	(* Internal method *)
	{attribute 'hide'}
	METHOD FB_init : BOOL
	VAR_INPUT
		(*  if TRUE, the retain variables are initialized (warm start / cold start) *)
		bInitRetains : BOOL;
		(*  if TRUE, the instance afterwards gets moved into the copy code (online change) *)
		bInCopyCode : BOOL;
	END_VAR
END_METHOD


	(* Internal method *)
	{attribute 'hide'}
	METHOD FB_exit : BOOL
	VAR_INPUT
		(*  if TRUE, the exit method is called for exiting an instance that is copied afterwards (online change). *)
		bInCopyCode : BOOL;
	END_VAR
END_METHOD


	(* Set the rotation angle in degrees [Â°]. *)
	METHOD SetAngle
	VAR_INPUT
		(* Rotation angle to set in degrees [Â°]. *)
		angle : LREAL;
	END_VAR
END_METHOD


	(* Set the components of this vector to '0.0'. *)
	METHOD SetZero
END_METHOD


	(* Set the components of this orientation. *)
	METHOD SetValues
	VAR_IN_OUT
		(* The position values to set. *)
 {attribute 'GUID' := '9769C204-E8C9-2F95-61E1-FD1671A2860B'}
				orientation2D : Orientation2D;
	END_VAR
END_METHOD


	(* Get the direction of the local x-axis. *)
	METHOD GetDirectionX
	VAR_IN_OUT
		(* The local x-direction of this orientation. *)
 {attribute 'GUID' := '5D3BC02D-EA16-22EA-7ADA-76A9B505DC98'}
				localX : TangentXY;
	END_VAR
END_METHOD


	(* Get the direction of the local y-axis. *)
	METHOD GetDirectionY
	VAR_IN_OUT
		(* The local y-direction of this orientation. *)
 {attribute 'GUID' := '5D3BC02D-EA16-22EA-7ADA-76A9B505DC98'}
				localY : TangentXY;
	END_VAR
END_METHOD


	(* Invert this position. *)
	METHOD Invert
END_METHOD


	(* Multiply an orientation to this orientation. *)
	METHOD ConcatenateWith
	VAR_IN_OUT
		(* Orientation to concatenate with. *)
 {attribute 'GUID' := '9769C204-E8C9-2F95-61E1-FD1671A2860B'}
				orientation2D : Orientation2D;
	END_VAR
END_METHOD


	(* Turn the orientation. *)
	METHOD TurnByC
	VAR_INPUT
		(* Rotation angle to turn by in degrees [Â°]. *)
		angle : LREAL;
	END_VAR
END_METHOD


	(* Rotate a PositionXY according to this orientation. *)
	METHOD Transform
	VAR_IN_OUT
		(* The orientation to multipy by. *)
 {attribute 'GUID' := 'ED71C9D8-8E4B-28CC-7DA0-249C4B114DE7'}
				positionXY : PositionXY;
	END_VAR
END_METHOD


	PROPERTY angle : LREAL
GET
END_GET
SET
END_SET
END_PROPERTY

END_FUNCTION_BLOCK

// POUs/Spatial/Functions/ConcatenateABC

	{attribute 'TcIecLibraryType'}
	{attribute 'external_name' := 'ConcatenateABC_GUID_63EF3EFF_CE46_22F7_7592_D84453B7BE61'}
	(* Concatenate two instances of Orientation3D. *)
	FUNCTION ConcatenateABC : BOOL
	VAR_IN_OUT
		rotation0	:	Orientation3D;	(* 1st input orientation of the concatenation. *)
		rotation1	:	Orientation3D;	(* 2nd input orientation of the concatenation. *)
		concatenation	:	Orientation3D;	(* The concatenation of the two input instances. *)
	END_VAR

END_FUNCTION

// POUs/Spatial/Positions/Orientation3D

	{attribute 'c++_compatible'}
	{attribute 'external_name' := 'Orientation3D_GUID_F3A50331_CB69_26F7_728F_6AA10FEBE6C7'}
	{attribute 'TcIecLibraryType'}
	{attribute 'no_explicit_call' :='do not call this POU directly'}
	{attribute 'no_assign'}
	(* 3D orientation. All angles in degrees [Â°]. *)
	FUNCTION_BLOCK Orientation3D
	VAR
		(* Rotation around the 1st local axis in degrees [Â°]. *)
		p0 : LREAL;
		(* Rotation around 2nd local axis in degrees [Â°]. *)
		p1 : LREAL;
		(* Rotation around 3rd local axis in degrees [Â°]. *)
		p2 : LREAL;
		(* Defines the rotation order (rotate around local axes from left to right) *)
		 {attribute 'GUID' := 'BF8BCC1E-925E-4A57-801C-CC42AFDDA86D'}
		coordinates : E_RotationCoordinates := E_RotationCoordinates.CBA;
		 {attribute 'hide'}
		_reserved1 : ARRAY [1..84] OF USINT;
	END_VAR


	(* Internal method *)
	{attribute 'hide'}
	METHOD FB_init : BOOL
	VAR_INPUT
		(*  if TRUE, the retain variables are initialized (warm start / cold start) *)
		bInitRetains : BOOL;
		(*  if TRUE, the instance afterwards gets moved into the copy code (online change) *)
		bInCopyCode : BOOL;
	END_VAR
END_METHOD


	(* Internal method *)
	{attribute 'hide'}
	METHOD FB_exit : BOOL
	VAR_INPUT
		(*  if TRUE, the exit method is called for exiting an instance that is copied afterwards (online change). *)
		bInCopyCode : BOOL;
	END_VAR
END_METHOD


	(* Set the components of this vector to '0.0'. *)
	METHOD SetZero
END_METHOD


	(* Set the components of this position. *)
	METHOD SetValues
	VAR_IN_OUT
		(* The position values to set. *)
 {attribute 'GUID' := 'F3A50331-CB69-26F7-728F-6AA10FEBE6C7'}
				orientation3D : Orientation3D;
	END_VAR
END_METHOD


	(* Set the coordinates of the orientation. *)
	METHOD SetValuesABC
	VAR_INPUT
		(* 1st rotation angle in degrees [Â°]. *)
		phi0 : LREAL;
		(* 2nd rotation angle in degrees [Â°]. *)
		phi1 : LREAL;
		(* 3rd rotation angle in degrees [Â°]. *)
		phi2 : LREAL;
	END_VAR
END_METHOD


	(* Set the coordinates of the orientation. *)
	METHOD SetValuesACB
	VAR_INPUT
		(* 1st rotation angle in degrees [Â°]. *)
		phi0 : LREAL;
		(* 2nd rotation angle in degrees [Â°]. *)
		phi1 : LREAL;
		(* 3rd rotation angle in degrees [Â°]. *)
		phi2 : LREAL;
	END_VAR
END_METHOD


	(* Set the coordinates of the orientation. *)
	METHOD SetValuesBCA
	VAR_INPUT
		(* 1st rotation angle in degrees [Â°]. *)
		phi0 : LREAL;
		(* 2nd rotation angle in degrees [Â°]. *)
		phi1 : LREAL;
		(* 3rd rotation angle in degrees [Â°]. *)
		phi2 : LREAL;
	END_VAR
END_METHOD


	(* Set the coordinates of the orientation. *)
	METHOD SetValuesBAC
	VAR_INPUT
		(* 1st rotation angle in degrees [Â°]. *)
		phi0 : LREAL;
		(* 2nd rotation angle in degrees [Â°]. *)
		phi1 : LREAL;
		(* 3rd rotation angle in degrees [Â°]. *)
		phi2 : LREAL;
	END_VAR
END_METHOD


	(* Set the coordinates of the orientation. *)
	METHOD SetValuesCAB
	VAR_INPUT
		(* 1st rotation angle in degrees [Â°]. *)
		phi0 : LREAL;
		(* 2nd rotation angle in degrees [Â°]. *)
		phi1 : LREAL;
		(* 3rd rotation angle in degrees [Â°]. *)
		phi2 : LREAL;
	END_VAR
END_METHOD


	(* Set the coordinates of the orientation. *)
	METHOD SetValuesCBA
	VAR_INPUT
		(* 1st rotation angle in degrees [Â°]. *)
		phi0 : LREAL;
		(* 2nd rotation angle in degrees [Â°]. *)
		phi1 : LREAL;
		(* 3rd rotation angle in degrees [Â°]. *)
		phi2 : LREAL;
	END_VAR
END_METHOD


	(* Set the coordinates of the orientation. *)
	METHOD SetValuesABA
	VAR_INPUT
		(* 1st rotation angle in degrees [Â°]. *)
		phi0 : LREAL;
		(* 2nd rotation angle in degrees [Â°]. *)
		phi1 : LREAL;
		(* 3rd rotation angle in degrees [Â°]. *)
		phi2 : LREAL;
	END_VAR
END_METHOD


	(* Set the coordinates of the orientation. *)
	METHOD SetValuesACA
	VAR_INPUT
		(* 1st rotation angle in degrees [Â°]. *)
		phi0 : LREAL;
		(* 2nd rotation angle in degrees [Â°]. *)
		phi1 : LREAL;
		(* 3rd rotation angle in degrees [Â°]. *)
		phi2 : LREAL;
	END_VAR
END_METHOD


	(* Set the coordinates of the orientation. *)
	METHOD SetValuesBCB
	VAR_INPUT
		(* 1st rotation angle in degrees [Â°]. *)
		phi0 : LREAL;
		(* 2nd rotation angle in degrees [Â°]. *)
		phi1 : LREAL;
		(* 3rd rotation angle in degrees [Â°]. *)
		phi2 : LREAL;
	END_VAR
END_METHOD


	(* Set the coordinates of the orientation. *)
	METHOD SetValuesBAB
	VAR_INPUT
		(* 1st rotation angle in degrees [Â°]. *)
		phi0 : LREAL;
		(* 2nd rotation angle in degrees [Â°]. *)
		phi1 : LREAL;
		(* 3rd rotation angle in degrees [Â°]. *)
		phi2 : LREAL;
	END_VAR
END_METHOD


	(* Set the coordinates of the orientation. *)
	METHOD SetValuesCAC
	VAR_INPUT
		(* 1st rotation angle in degrees [Â°]. *)
		phi0 : LREAL;
		(* 2nd rotation angle in degrees [Â°]. *)
		phi1 : LREAL;
		(* 3rd rotation angle in degrees [Â°]. *)
		phi2 : LREAL;
	END_VAR
END_METHOD


	(* Set the coordinates of the orientation. *)
	METHOD SetValuesCBC
	VAR_INPUT
		(* 1st rotation angle in degrees [Â°]. *)
		phi0 : LREAL;
		(* 2nd rotation angle in degrees [Â°]. *)
		phi1 : LREAL;
		(* 3rd rotation angle in degrees [Â°]. *)
		phi2 : LREAL;
	END_VAR
END_METHOD


	(* Get the direction of the local x-axis. *)
	METHOD GetDirectionX
	VAR_IN_OUT
		(* The local x-direction of this orientation. *)
 {attribute 'GUID' := '8E451EF0-1EF7-2C22-40FE-C3C408FD9C3F'}
				localX : Tangent3D;
	END_VAR
END_METHOD


	(* Get the direction of the local y-axis. *)
	METHOD GetDirectionY
	VAR_IN_OUT
		(* The local y-direction of this orientation. *)
 {attribute 'GUID' := '8E451EF0-1EF7-2C22-40FE-C3C408FD9C3F'}
				localY : Tangent3D;
	END_VAR
END_METHOD


	(* Get the direction of the local z-axis. *)
	METHOD GetDirectionZ
	VAR_IN_OUT
		(* The local z-direction of this orientation. *)
 {attribute 'GUID' := '8E451EF0-1EF7-2C22-40FE-C3C408FD9C3F'}
				localZ : Tangent3D;
	END_VAR
END_METHOD


	(* Invert this position. *)
	METHOD Invert
END_METHOD


	(* Multiply an orientation to this orientation. *)
	METHOD ConcatenateWith
	VAR_IN_OUT
		(* Orientation to concatenate with. *)
 {attribute 'GUID' := 'F3A50331-CB69-26F7-728F-6AA10FEBE6C7'}
				orientation : Orientation3D;
	END_VAR
END_METHOD


	(* Rotate around an arbitrary local axis. The turn angle is given by the length of the axis. *)
	METHOD TurnBy
	VAR_IN_OUT
		(* The axis of rotation. Its length represents the angle of rotation in degrees [Â°]. *)
 {attribute 'GUID' := '7C1DEECE-32AB-2E94-7A82-2C8AD444717E'}
				axis : TangentABC;
	END_VAR
END_METHOD


	(* Rotation around the local x-axis. *)
	METHOD TurnByA
	VAR_INPUT
		(* The angle to rotate by in degrees [Â°]. *)
		da : LREAL;
	END_VAR
END_METHOD


	(* Rotation around the local y-axis. *)
	METHOD TurnByB
	VAR_INPUT
		(* The angle to rotate by in degrees [Â°]. *)
		db : LREAL;
	END_VAR
END_METHOD


	(* Rotation around the local z-axis. *)
	METHOD TurnByC
	VAR_INPUT
		(* The angle to rotate by in degrees [Â°]. *)
		dc : LREAL;
	END_VAR
END_METHOD


	(* Rotate a Position3D according to this orientation. *)
	METHOD Transform
	VAR_IN_OUT
		(* Position to transform. *)
 {attribute 'GUID' := '513B7ECA-E1D5-262C-5763-788E1FD4F5AD'}
				position3D : Position3D;
	END_VAR
END_METHOD


	PROPERTY phi0 : LREAL
GET
END_GET
SET
END_SET
END_PROPERTY


	PROPERTY phi1 : LREAL
GET
END_GET
SET
END_SET
END_PROPERTY


	PROPERTY phi2 : LREAL
GET
END_GET
SET
END_SET
END_PROPERTY


	PROPERTY convention : E_RotationCoordinates
GET
END_GET
SET
END_SET
END_PROPERTY

END_FUNCTION_BLOCK

// POUs/Spatial/Functions/ConcatenateXYC

	{attribute 'TcIecLibraryType'}
	{attribute 'external_name' := 'ConcatenateXYC_GUID_447068A6_9467_2251_75A9_C1FF62E2E084'}
	(* Concatenate two instances of PositionXYC. *)
	FUNCTION ConcatenateXYC : BOOL
	VAR_IN_OUT
		position0	:	PositionXYC;	(* 1st input position of the concatenation. *)
		position1	:	PositionXYC;	(* 2nd input position of the concatenation. *)
		concatenation	:	PositionXYC;	(* The concatenation of the two input instances. *)
	END_VAR

END_FUNCTION

// POUs/Spatial/Functions/Concatenate6D

	{attribute 'TcIecLibraryType'}
	{attribute 'external_name' := 'Concatenate6D_GUID_B218722C_9A1D_2627_473C_2033807B3EB5'}
	(* Concatenate two instances of PositionSE3. *)
	FUNCTION Concatenate6D : BOOL
	VAR_IN_OUT
		position0	:	PositionSE3;	(* 1st input position of the concatenation. *)
		position1	:	PositionSE3;	(* 2nd input position of the concatenation. *)
		concatenation	:	PositionXYC;	(* The concatenation of the two input instances. *)
	END_VAR

END_FUNCTION

// POUs/Spatial/Functions/AddXY

	{attribute 'TcIecLibraryType'}
	{attribute 'external_name' := 'AddXY_GUID_E175C5D9_61B7_2C72_416A_96A339F4B43B'}
	(* Add two instances of TangentXY. *)
	FUNCTION AddXY : BOOL
	VAR_IN_OUT
		tangent0	:	TangentXY;	(* 1st input tangent vector. *)
		tangent1	:	TangentXY;	(* 2nd input tangent vector. *)
		sumTangent	:	TangentXY;	(* Sum of the two tangent vectors. *)
	END_VAR

END_FUNCTION

// POUs/Spatial/Functions/SubtractXY

	{attribute 'TcIecLibraryType'}
	{attribute 'external_name' := 'SubtractXY_GUID_30C9C628_6AA3_2EA8_7056_6D631FEDD6CC'}
	(* Subtract two instances of TangentXY. *)
	FUNCTION SubtractXY : BOOL
	VAR_IN_OUT
		tangent0	:	TangentXY;	(* 1st input tangent vector. *)
		tangent1	:	TangentXY;	(* 2nd input tangent vector. *)
		difference	:	TangentXY;	(* Difference of the two tangent vectors. *)
	END_VAR

END_FUNCTION

// POUs/Spatial/Functions/MultiplyXY

	{attribute 'TcIecLibraryType'}
	{attribute 'external_name' := 'MultiplyXY_GUID_FE62303C_7D56_2E0D_77DF_EC3A00A94E9C'}
	(* Multiply a TangentXY by a scalar and return the result. *)
	FUNCTION MultiplyXY : BOOL
	VAR_IN_OUT
		tangent	:	TangentXY;	(* Tangent vector to multiply. *)
	END_VAR
	VAR_INPUT
		scalar	:	LREAL;	(* Scalar value to multiply with. *)
	END_VAR
	VAR_IN_OUT
		scaled	:	TangentXY;	(* Scaled input tangent vector. *)
	END_VAR

END_FUNCTION

// POUs/Spatial/Functions/ScalarXY

	{attribute 'TcIecLibraryType'}
	{attribute 'external_name' := 'ScalarXY_GUID_E87FF040_9366_28D4_7F75_DB012A742D5B'}
	(* Compute the scalar product of two instance of TangentXY. *)
	FUNCTION ScalarXY : LREAL
	VAR_IN_OUT
		tangent0	:	TangentXY;	(* 1st input tangent vector. *)
		tangent1	:	TangentXY;	(* 2nd input tangent vector. *)
	END_VAR

END_FUNCTION

// POUs/Spatial/Functions/Add3D

	{attribute 'TcIecLibraryType'}
	{attribute 'external_name' := 'Add3D_GUID_22B5713A_DAAE_208F_5845_FFB0DA8961E0'}
	(* Add two instances of Tangent3D. *)
	FUNCTION Add3D : BOOL
	VAR_IN_OUT
		tangent0	:	Tangent3D;	(* 1st input tangent vector. *)
		tangent1	:	Tangent3D;	(* 2nd input tangent vector. *)
		sumTangent	:	Tangent3D;	(* Sum of the two tangent vectors. *)
	END_VAR

END_FUNCTION

// POUs/Spatial/Functions/Subtract3D

	{attribute 'TcIecLibraryType'}
	{attribute 'external_name' := 'Subtract3D_GUID_3F13D96E_61B4_2521_768F_ABB3A2BB8B32'}
	(* Subtract two instances of Tangent3D. *)
	FUNCTION Subtract3D : BOOL
	VAR_IN_OUT
		tangent0	:	Tangent3D;	(* 1st input tangent vector. *)
		tangent1	:	Tangent3D;	(* 2nd input tangent vector. *)
		difference	:	Tangent3D;	(* Difference of the two tangent vectors. *)
	END_VAR

END_FUNCTION

// POUs/Spatial/Functions/Multiply3D

	{attribute 'TcIecLibraryType'}
	{attribute 'external_name' := 'Multiply3D_GUID_43B67DFD_6BDE_217D_78F1_09963C777F30'}
	(* Multiply a Tangent3D by a scalar. *)
	FUNCTION Multiply3D : BOOL
	VAR_IN_OUT
		tangent	:	Tangent3D;	(* Tangent vector to multiply. *)
	END_VAR
	VAR_INPUT
		scalar	:	LREAL;	(* Scalar value to multiply with. *)
	END_VAR
	VAR_IN_OUT
		scaled	:	Tangent3D;	(* Scaled input tangent vector. *)
	END_VAR

END_FUNCTION

// POUs/Spatial/Functions/Scalar3D

	{attribute 'TcIecLibraryType'}
	{attribute 'external_name' := 'Scalar3D_GUID_B656DD08_36BC_2264_65B8_8E86D53E44D8'}
	(* Compute the scalar product of two instances of Tangent3D. *)
	FUNCTION Scalar3D : LREAL
	VAR_IN_OUT
		tangent0	:	Tangent3D;	(* 1st input tangent vector. *)
		tangent1	:	Tangent3D;	(* 2nd input tangent vector. *)
	END_VAR

END_FUNCTION

// POUs/Spatial/Functions/Cross3D

	{attribute 'TcIecLibraryType'}
	{attribute 'external_name' := 'Cross3D_GUID_637E2F8F_7C67_21A9_5D9B_C69EDB5530E5'}
	(* Compute the cross product of two instances of Tangent3D. *)
	FUNCTION Cross3D : BOOL
	VAR_IN_OUT
		tangent0	:	Tangent3D;	(* 1st input tangent vector. *)
		tangent1	:	Tangent3D;	(* 2nd input tangent vector. *)
		crossProduct	:	Tangent3D;	(* The resulting cross product. *)
	END_VAR

END_FUNCTION

// POUs/Spatial/Functions/AddABC

	{attribute 'TcIecLibraryType'}
	{attribute 'external_name' := 'AddABC_GUID_B378EB54_DC30_2FB7_4703_748A68BC554E'}
	(* Add two instances of TangentABC. *)
	FUNCTION AddABC : BOOL
	VAR_IN_OUT
		tangent0	:	TangentABC;	(* 1st input tangent vector. *)
		tangent1	:	TangentABC;	(* 2nd input tangent vector. *)
		sumTangent	:	TangentABC;	(* Sum of the two tangent vectors. *)
	END_VAR

END_FUNCTION

// POUs/Spatial/Functions/SubtractABC

	{attribute 'TcIecLibraryType'}
	{attribute 'external_name' := 'SubtractABC_GUID_0EC77355_F7D6_2D64_72F6_4550677466CB'}
	(* Subtract two instances of TangentABC. *)
	FUNCTION SubtractABC : BOOL
	VAR_IN_OUT
		tangent0	:	TangentABC;	(* 1st input tangent vector. *)
		tangent1	:	TangentABC;	(* 2nd input tangent vector. *)
		difference	:	TangentABC;	(* Difference of the two tangent vectors. *)
	END_VAR

END_FUNCTION

// POUs/Spatial/Functions/MultiplyABC

	{attribute 'TcIecLibraryType'}
	{attribute 'external_name' := 'MultiplyABC_GUID_CED5725A_0908_2221_656C_470734809FE5'}
	(* Multiply a TangentABC by a scalar. *)
	FUNCTION MultiplyABC : BOOL
	VAR_IN_OUT
		tangent	:	TangentABC;	(* Tangent vector to multiply. *)
	END_VAR
	VAR_INPUT
		scalar	:	LREAL;	(* Scalar value to multiply with. *)
	END_VAR
	VAR_IN_OUT
		scaled	:	TangentABC;	(* Scaled input tangent vector. *)
	END_VAR

END_FUNCTION

// POUs/Spatial/Functions/AddXYC

	{attribute 'TcIecLibraryType'}
	{attribute 'external_name' := 'AddXYC_GUID_1E14462F_988B_29BB_78EF_085C7340C86C'}
	(* Add two instances of TangentXYC. *)
	FUNCTION AddXYC : BOOL
	VAR_IN_OUT
		tangent0	:	TangentXYC;	(* 1st input tangent vector. *)
		tangent1	:	TangentXYC;	(* 2nd input tangent vector. *)
		sumTangent	:	TangentXYC;	(* Sum of the two tangent vectors. *)
	END_VAR

END_FUNCTION

// POUs/Spatial/Functions/SubtractXYC

	{attribute 'TcIecLibraryType'}
	{attribute 'external_name' := 'SubtractXYC_GUID_DDE910B0_CB45_27E1_47FA_8B6FC171A22B'}
	(* Subtract two instances of TangentXYC. *)
	FUNCTION SubtractXYC : BOOL
	VAR_IN_OUT
		tangent0	:	TangentXYC;	(* 1st input tangent vector. *)
		tangent1	:	TangentXYC;	(* 2nd input tangent vector. *)
		difference	:	TangentXYC;	(* Difference of the two tangent vectors. *)
	END_VAR

END_FUNCTION

// POUs/Spatial/Functions/MultiplyXYC

	{attribute 'TcIecLibraryType'}
	{attribute 'external_name' := 'MultiplyXYC_GUID_6B3384A2_CB86_2C92_42CE_70FAA85DA471'}
	(* Multiply a TangentXYC by a scalar. *)
	FUNCTION MultiplyXYC : BOOL
	VAR_IN_OUT
		tangent	:	TangentXYC;	(* Tangent vector to multiply. *)
	END_VAR
	VAR_INPUT
		scalar	:	LREAL;	(* Scalar value to multiply with. *)
	END_VAR
	VAR_IN_OUT
		scaled	:	TangentXYC;	(* Scaled input tangent vector. *)
	END_VAR

END_FUNCTION

// POUs/Spatial/Functions/Add6D

	{attribute 'TcIecLibraryType'}
	{attribute 'external_name' := 'Add6D_GUID_0B14101C_9D2D_2597_7509_08E24C33C593'}
	(* Add two instances of Tangent6D. *)
	FUNCTION Add6D : BOOL
	VAR_IN_OUT
		tangent0	:	Tangent6D;	(* 1st input tangent vector. *)
		tangent1	:	Tangent6D;	(* 2nd input tangent vector. *)
		sumTangent	:	Tangent6D;	(* Sum of the two tangent vectors. *)
	END_VAR

END_FUNCTION

// POUs/Spatial/Functions/Subtract6D

	{attribute 'TcIecLibraryType'}
	{attribute 'external_name' := 'Subtract6D_GUID_FE876AD6_8028_2A78_507A_F5438F4E99D8'}
	(* Subtract two instances of Tangent6D. *)
	FUNCTION Subtract6D : BOOL
	VAR_IN_OUT
		tangent0	:	Tangent6D;	(* 1st input tangent vector. *)
		tangent1	:	Tangent6D;	(* 2nd input tangent vector. *)
		difference	:	Tangent6D;	(* Difference of the two tangent vectors. *)
	END_VAR

END_FUNCTION

// POUs/Spatial/Functions/Multiply6D

	{attribute 'TcIecLibraryType'}
	{attribute 'external_name' := 'Multiply6D_GUID_EADA0247_E296_2995_4AF7_01DD583E2BDC'}
	(* Multiply a Tangent6D by a scalar. *)
	FUNCTION Multiply6D : BOOL
	VAR_IN_OUT
		tangent	:	Tangent6D;	(* Tangent vector to multiply. *)
	END_VAR
	VAR_INPUT
		scalar	:	LREAL;	(* Scalar value to multiply with. *)
	END_VAR
	VAR_IN_OUT
		scaled	:	Tangent6D;	(* Scaled input tangent vector. *)
	END_VAR

END_FUNCTION

// POUs/Spatial/Functions/ConvertToCartesian2D

	{attribute 'TcIecLibraryType'}
	{attribute 'external_name' := 'ConvertToCartesian2D_GUID_66635609_EA9D_20E7_752F_19ECB689283F'}
	(* Convert local XYC-dynamic properties to global XY ones. *)
	FUNCTION ConvertToCartesian2D : BOOL
	VAR_IN_OUT
		position	:	PositionXYC;	(* The position hosting the local dynamic state. *)
		velocity	:	TangentXYC;	(* The local velocity vector. *)
		acceleration	:	TangentXYC;	(* The local acceleration vector. *)
		velocity_XY	:	TangentXY;	(* The resulting global Cartesian velocity. *)
		acceleration_XY	:	TangentXY;	(* The resulting global Cartesian acceleration. *)
	END_VAR

END_FUNCTION

// POUs/Spatial/Setpoints/SetpointR1

	{attribute 'c++_compatible'}
	{attribute 'external_name' := 'SetpointR1_GUID_377B7699_EBC9_237A_45F1_345E01A5B7D6'}
	{attribute 'TcIecLibraryType'}
	{attribute 'no_explicit_call' :='do not call this POU directly'}
	{attribute 'no_assign_warning'}
	(* 1D setpoint. *)
	FUNCTION_BLOCK SetpointR1
	VAR
		(* Position component of the setpoint. *)
		ds : LREAL;
		(* Velocity component of the setpoint. *)
		dv : LREAL;
		(* Acceleration component of the setpoint. *)
		da : LREAL;
		(* Jerk component of the setpoint. *)
		dj : LREAL;
	END_VAR


	(* Internal method *)
	{attribute 'hide'}
	METHOD FB_init : BOOL
	VAR_INPUT
		(*  if TRUE, the retain variables are initialized (warm start / cold start) *)
		bInitRetains : BOOL;
		(*  if TRUE, the instance afterwards gets moved into the copy code (online change) *)
		bInCopyCode : BOOL;
	END_VAR
END_METHOD


	(* Internal method *)
	{attribute 'hide'}
	METHOD FB_reinit : BOOL
END_METHOD


	(* Internal method *)
	{attribute 'hide'}
	METHOD FB_exit : BOOL
	VAR_INPUT
		(*  if TRUE, the exit method is called for exiting an instance that is copied afterwards (online change). *)
		bInCopyCode : BOOL;
	END_VAR
END_METHOD


	(* Set this setpoint to zero. *)
	METHOD SetZero
END_METHOD


	(* Set the values of this coordinate. *)
	METHOD SetValuesSVAJ
	VAR_INPUT
		(* the position value to set. *)
		_s : LREAL;
		(* the velocity value to set. *)
		v : LREAL;
		(* the acceleration value to set. *)
		a : LREAL;
		(* the jerk value to set. *)
		j : LREAL;
	END_VAR
END_METHOD


	PROPERTY _s : LREAL
GET
END_GET
SET
END_SET
END_PROPERTY


	PROPERTY v : LREAL
GET
END_GET
SET
END_SET
END_PROPERTY


	PROPERTY a : LREAL
GET
END_GET
SET
END_SET
END_PROPERTY


	PROPERTY j : LREAL
GET
END_GET
SET
END_SET
END_PROPERTY

END_FUNCTION_BLOCK

// POUs/Spatial/Setpoints/SetpointSE3

	{attribute 'c++_compatible'}
	{attribute 'external_name' := 'SetpointSE3_GUID_A3F4D6D1_1484_2B13_6519_BC8D5184F1A9'}
	{attribute 'TcIecLibraryType'}
	{attribute 'no_explicit_call' :='do not call this POU directly'}
	{attribute 'no_assign_warning'}
	(* SE3 setpoint. *)
	FUNCTION_BLOCK SetpointSE3 EXTENDS IPlcGeometry3D


	(* Internal method *)
	{attribute 'hide'}
	METHOD FB_init : BOOL
	VAR_INPUT
		(*  if TRUE, the retain variables are initialized (warm start / cold start) *)
		bInitRetains : BOOL;
		(*  if TRUE, the instance afterwards gets moved into the copy code (online change) *)
		bInCopyCode : BOOL;
	END_VAR
END_METHOD


	(* Internal method *)
	{attribute 'hide'}
	METHOD FB_exit : BOOL
	VAR_INPUT
		(*  if TRUE, the exit method is called for exiting an instance that is copied afterwards (online change). *)
		bInCopyCode : BOOL;
	END_VAR
END_METHOD


	(* Set this setpoint to be the identity. *)
	METHOD SetIdentity
END_METHOD


	(* Set the values of this setpoint. *)
	METHOD SetValues
	VAR_IN_OUT
		(* The setpoint to copy. *)
 {attribute 'GUID' := 'A3F4D6D1-1484-2B13-6519-BC8D5184F1A9'}
				setpoint : SetpointSE3;
	END_VAR
END_METHOD


	(* Set the cartesian values of this setpoint. *)
	METHOD SetValuesXYZ
	VAR_IN_OUT
		(* The x-setpoint to set. *)
 {attribute 'GUID' := '377B7699-EBC9-237A-45F1-345E01A5B7D6'}
				setpointX : SetpointR1;
		(* The y-setpoint to set. *)
 {attribute 'GUID' := '377B7699-EBC9-237A-45F1-345E01A5B7D6'}
				setpointY : SetpointR1;
		(* The z-setpoint to set. *)
 {attribute 'GUID' := '377B7699-EBC9-237A-45F1-345E01A5B7D6'}
				setpointZ : SetpointR1;
	END_VAR
END_METHOD


	(* Set the angular values of this setpoint. *)
	METHOD SetValuesCBA
	VAR_IN_OUT
		(* The c-setpoint to set. *)
 {attribute 'GUID' := '377B7699-EBC9-237A-45F1-345E01A5B7D6'}
				setpointC : SetpointR1;
		(* The b-setpoint to set. *)
 {attribute 'GUID' := '377B7699-EBC9-237A-45F1-345E01A5B7D6'}
				setpointB : SetpointR1;
		(* The a-setpoint to set. *)
 {attribute 'GUID' := '377B7699-EBC9-237A-45F1-345E01A5B7D6'}
				setpointA : SetpointR1;
	END_VAR
END_METHOD


	(* Get the direction of the local x-axis. *)
	METHOD GetDirectionX
	VAR_IN_OUT
		(* The local x-direction of this orientation. *)
 {attribute 'GUID' := '8E451EF0-1EF7-2C22-40FE-C3C408FD9C3F'}
				localX : Tangent3D;
	END_VAR
END_METHOD


	(* Get the direction of the local y-axis. *)
	METHOD GetDirectionY
	VAR_IN_OUT
		(* The local y-direction of this orientation. *)
 {attribute 'GUID' := '8E451EF0-1EF7-2C22-40FE-C3C408FD9C3F'}
				localY : Tangent3D;
	END_VAR
END_METHOD


	(* Get the direction of the local z-axis. *)
	METHOD GetDirectionZ
	VAR_IN_OUT
		(* The local z-direction of this orientation. *)
 {attribute 'GUID' := '8E451EF0-1EF7-2C22-40FE-C3C408FD9C3F'}
				localZ : Tangent3D;
	END_VAR
END_METHOD


	(* Get the linear Cartesian position components. *)
	METHOD GetPosition_Cartesian
	VAR_IN_OUT
		(* The output position. *)
 {attribute 'GUID' := '513B7ECA-E1D5-262C-5763-788E1FD4F5AD'}
				position : Position3D;
	END_VAR
END_METHOD


	(* Get the linear Cartesian velocity components. *)
	METHOD GetVelocity_Cartesian
	VAR_IN_OUT
		(* The output tangent. *)
 {attribute 'GUID' := '8E451EF0-1EF7-2C22-40FE-C3C408FD9C3F'}
				tangent : Tangent3D;
	END_VAR
END_METHOD


	(* Get the linear Cartesian acceleration components. *)
	METHOD GetAcceleration_Cartesian
	VAR_IN_OUT
		(* The output tangent. *)
 {attribute 'GUID' := '8E451EF0-1EF7-2C22-40FE-C3C408FD9C3F'}
				tangent : Tangent3D;
	END_VAR
END_METHOD


	(* Get the linear Cartesian jerk components. *)
	METHOD GetJerk_Cartesian
	VAR_IN_OUT
		(* The output tangent. *)
 {attribute 'GUID' := '8E451EF0-1EF7-2C22-40FE-C3C408FD9C3F'}
				tangent : Tangent3D;
	END_VAR
END_METHOD


	(* Concatenate this setpoint with a second one up to a specific order. *)
	METHOD ConcatenateWith
	VAR_IN_OUT
		(* The setpoint to concatenate. *)
 {attribute 'GUID' := 'A3F4D6D1-1484-2B13-6519-BC8D5184F1A9'}
				setpoint : SetpointSE3;
	END_VAR
	VAR_INPUT
		(*  The order up to which to compute. *)
		order : UDINT;
	END_VAR
END_METHOD


	PROPERTY x : LREAL
GET
END_GET
SET
END_SET
END_PROPERTY


	PROPERTY y : LREAL
GET
END_GET
SET
END_SET
END_PROPERTY


	PROPERTY z : LREAL
GET
END_GET
SET
END_SET
END_PROPERTY


	PROPERTY phi0 : LREAL
GET
END_GET
SET
END_SET
END_PROPERTY


	PROPERTY phi1 : LREAL
GET
END_GET
SET
END_SET
END_PROPERTY


	PROPERTY phi2 : LREAL
GET
END_GET
SET
END_SET
END_PROPERTY


	PROPERTY Convention : E_RotationCoordinates
GET
END_GET
SET
END_SET
END_PROPERTY

END_FUNCTION_BLOCK

// POUs/Spatial/Inertias/InertiaSE3

	{attribute 'c++_compatible'}
	{attribute 'external_name' := 'InertiaSE3_GUID_3BA5DEBC_CD81_22A1_4AA7_D2CA603D8F2C'}
	{attribute 'TcIecLibraryType'}
	{attribute 'no_explicit_call' :='do not call this POU directly'}
	{attribute 'no_assign'}
	(* Inertia tensor containing angular and linear inertia. *)
	FUNCTION_BLOCK InertiaSE3
	VAR
		(* Mass of the inertia. *)
		m : LREAL;
		(* x-component of the center of mass. *)
		CenterX : LREAL;
		(* y-component of the center of mass. *)
		CenterY : LREAL;
		(* z-component of the center of mass. *)
		CenterZ : LREAL;
		 {attribute 'hide'}
		_reserved1 : ARRAY [1..80] OF USINT;
	END_VAR


	(* Internal method *)
	{attribute 'hide'}
	METHOD FB_init : BOOL
	VAR_INPUT
		(*  if TRUE, the retain variables are initialized (warm start / cold start) *)
		bInitRetains : BOOL;
		(*  if TRUE, the instance afterwards gets moved into the copy code (online change) *)
		bInCopyCode : BOOL;
	END_VAR
END_METHOD


	(* Internal method *)
	{attribute 'hide'}
	METHOD FB_exit : BOOL
	VAR_INPUT
		(*  if TRUE, the exit method is called for exiting an instance that is copied afterwards (online change). *)
		bInCopyCode : BOOL;
	END_VAR
END_METHOD


	(* Add a 2nd inertia tensor to this one. *)
	METHOD AddBy
	VAR_IN_OUT
		(* The inertia tensor to add. *)
 {attribute 'GUID' := '3BA5DEBC-CD81-22A1-4AA7-D2CA603D8F2C'}
				shift : InertiaSE3;
	END_VAR
END_METHOD


	(* Set the values to that of a point. *)
	METHOD SetValues_Point
	VAR_INPUT
		(* The mass of the point. *)
		mass : LREAL;
		(* The x-position of the point. *)
		x : LREAL;
		(* The y-position of the point. *)
		y : LREAL;
		(* The z-position of the point. *)
		z : LREAL;
	END_VAR
END_METHOD


	(* Set the values to that of a sphere. *)
	METHOD SetValues_Sphere
	VAR_INPUT
		(* The mass of the sphere. *)
		mass : LREAL;
		(* The radius of the sphere. *)
		radius : LREAL;
	END_VAR
END_METHOD


	(* Set the values to that of a cylinder. *)
	METHOD SetValues_Cylinder
	VAR_INPUT
		(* The mass of the cylinder. *)
		mass : LREAL;
		(* The radius of the cylinder. *)
		radius : LREAL;
		(* The height of the cylinder. *)
		height : LREAL;
	END_VAR
END_METHOD


	(* Set the values to that of a cuboid. *)
	METHOD SetValues_Cuboid
	VAR_INPUT
		(* The mass of the cuboid. *)
		mass : LREAL;
		(* The x-length of the cuboid. *)
		dx : LREAL;
		(* The y-length of the cuboid. *)
		dy : LREAL;
		(* The z-length of the cuboid. *)
		dz : LREAL;
	END_VAR
END_METHOD


	(* Transform this inertia by a displacement. *)
	METHOD Transform
	VAR_IN_OUT
		(* The displacement to apply. *)
 {attribute 'GUID' := '71570C9B-708B-2C60-4B94-668F28922D38'}
				displacement : PositionSE3;
	END_VAR
END_METHOD


	(* Translate this inertia by a translation. *)
	METHOD Translate
	VAR_IN_OUT
		(* The translation to apply. *)
 {attribute 'GUID' := '8E451EF0-1EF7-2C22-40FE-C3C408FD9C3F'}
				displacement : Tangent3D;
	END_VAR
END_METHOD


	PROPERTY mass : LREAL
GET
END_GET
SET
END_SET
END_PROPERTY


	PROPERTY x : LREAL
GET
END_GET
SET
END_SET
END_PROPERTY


	PROPERTY y : LREAL
GET
END_GET
SET
END_SET
END_PROPERTY


	PROPERTY z : LREAL
GET
END_GET
SET
END_SET
END_PROPERTY


	PROPERTY xx : LREAL
GET
END_GET
SET
END_SET
END_PROPERTY


	PROPERTY yy : LREAL
GET
END_GET
SET
END_SET
END_PROPERTY


	PROPERTY zz : LREAL
GET
END_GET
SET
END_SET
END_PROPERTY


	PROPERTY xy : LREAL
GET
END_GET
SET
END_SET
END_PROPERTY


	PROPERTY yz : LREAL
GET
END_GET
SET
END_SET
END_PROPERTY


	PROPERTY zx : LREAL
GET
END_GET
SET
END_SET
END_PROPERTY

END_FUNCTION_BLOCK

// POUs/Shapes/Geometry2D/Container2D

	{attribute 'c++_compatible'}
	{attribute 'external_name' := 'Container2D_GUID_4AD80F83_4F38_2FF8_4DD5_6F1BB78BF649'}
	{attribute 'TcIecLibraryType'}
	{attribute 'no_explicit_call' :='do not call this POU directly'}
	{attribute 'no_assign'}
	FUNCTION_BLOCK Container2D EXTENDS Geometry2D


	(* Internal method *)
	METHOD FB_init : BOOL
	VAR_INPUT
		(*  if TRUE, the retain variables are initialized (warm start / cold start) *)
		bInitRetains : BOOL;
		(*  if TRUE, the instance afterwards gets moved into the copy code (online change) *)
		bInCopyCode : BOOL;
	END_VAR
END_METHOD


	(* Internal method *)
	{attribute 'hide'}
	METHOD FB_exit : BOOL
	VAR_INPUT
		(*  if TRUE, the exit method is called for exiting an instance that is copied afterwards (online change). *)
		bInCopyCode : BOOL;
	END_VAR
END_METHOD


	(* Add a geometry to the container. *)
	METHOD AddElement : UDINT
	VAR_IN_OUT
		(* The geometry to add. *)
 {attribute 'GUID' := 'D6BFB8FE-9CFD-26BE-6EA3-D763AD2569A4'}
				inputObject : Geometry2D;
	END_VAR
END_METHOD


	(* Remove a specified geometry from the container. *)
	METHOD RemoveElement
	VAR_INPUT
		(* ID of the geometry to remove. *)
		id : UDINT;
	END_VAR
END_METHOD


	(* Remove all geometries from the container. *)
	METHOD Clear
END_METHOD


	(* Get the number of geometry elements in container. *)
	METHOD GetCount : UDINT
END_METHOD


	(* Get the combined boundary of all hosted 2D-geometries. *)
	METHOD GetBoundary
	VAR_IN_OUT
		(* The combined boundary.. *)
 {attribute 'GUID' := '4AD80F83-4F38-2FF8-4DD5-6F1BB78BF649'}
				boundary : Container2D;
	END_VAR
END_METHOD

END_FUNCTION_BLOCK

// POUs/Shapes/Geometry2D/Extrude2D

	{attribute 'c++_compatible'}
	{attribute 'external_name' := 'Extrude2D_GUID_DCBA8928_B44D_2C41_43DF_F3E6236BA280'}
	{attribute 'TcIecLibraryType'}
	{attribute 'no_explicit_call' :='do not call this POU directly'}
	{attribute 'no_assign'}
	FUNCTION_BLOCK Extrude2D EXTENDS Geometry2D


	(* Internal method *)
	METHOD FB_init : BOOL
	VAR_INPUT
		(*  if TRUE, the retain variables are initialized (warm start / cold start) *)
		bInitRetains : BOOL;
		(*  if TRUE, the instance afterwards gets moved into the copy code (online change) *)
		bInCopyCode : BOOL;
	END_VAR
END_METHOD


	(* Internal method *)
	{attribute 'hide'}
	METHOD FB_exit : BOOL
	VAR_INPUT
		(*  if TRUE, the exit method is called for exiting an instance that is copied afterwards (online change). *)
		bInCopyCode : BOOL;
	END_VAR
END_METHOD


	(* Define the extrusion geometry by a path and the corners to extrude. *)
	METHOD ExtrudeAlong
	VAR_IN_OUT
		(* The path to extrude along. *)
 {attribute 'GUID' := '7FCF97B8-20CD-2CA3-6B3F-E4AF29A0B8D7'}
				path : PathXYC;
	END_VAR
	VAR_INPUT
		(* 1st distance from the path to extrude. *)
		dy0 : LREAL;
		(* 2nd distance from the path to extrude. *)
		dy1 : LREAL;
		(* Number of steps to employ along the path. *)
		extrusionSteps : UDINT;
	END_VAR
END_METHOD


	(* Check whether this extrusion geometry is valid. *)
	METHOD IsValid : BOOL
END_METHOD

END_FUNCTION_BLOCK

// POUs/Paths/Components/PathXYC

	{attribute 'c++_compatible'}
	{attribute 'external_name' := 'PathXYC_GUID_7FCF97B8_20CD_2CA3_6B3F_E4AF29A0B8D7'}
	{attribute 'TcIecLibraryType'}
	{attribute 'no_explicit_call' :='do not call this POU directly'}
	{attribute 'no_assign'}
	(* A path in the xy-plane with an additional orientation at every path position. *)
	FUNCTION_BLOCK PathXYC EXTENDS IPlcPath2D


	(* Internal method *)
	{attribute 'hide'}
	METHOD FB_init : BOOL
	VAR_INPUT
		(*  if TRUE, the retain variables are initialized (warm start / cold start) *)
		bInitRetains : BOOL;
		(*  if TRUE, the instance afterwards gets moved into the copy code (online change) *)
		bInCopyCode : BOOL;
	END_VAR
END_METHOD


	(* Internal method *)
	{attribute 'hide'}
	METHOD FB_exit : BOOL
	VAR_INPUT
		(*  if TRUE, the exit method is called for exiting an instance that is copied afterwards (online change). *)
		bInCopyCode : BOOL;
	END_VAR
END_METHOD


	(* Append a smooth transition from the current end of the path
				    to the specified position. *)
	METHOD AppendPosition
	VAR_IN_OUT
		(* The position to append. *)
 {attribute 'GUID' := '684B7065-E3A9-208A-688F-6768C580A855'}
				position : PositionXYC;
	END_VAR
END_METHOD


	(* Append a smooth transition from the current end of the path
				    to the specified position. *)
	METHOD AppendPositionXYC
	VAR_INPUT
		(* x-component of the position to append. *)
		x : LREAL;
		(* y-component of the position to append. *)
		y : LREAL;
		(* c-component of the position to append in degrees [Â°]. *)
		c : LREAL;
	END_VAR
END_METHOD


	(* Append a line to this path. *)
	METHOD AppendLine
	VAR_IN_OUT
		(* Start position of the line. *)
 {attribute 'GUID' := '684B7065-E3A9-208A-688F-6768C580A855'}
				startPos : PositionXYC;
		(* End position of the line. *)
 {attribute 'GUID' := '684B7065-E3A9-208A-688F-6768C580A855'}
				endPos : PositionXYC;
	END_VAR
END_METHOD


	(* Append a circle to this path. *)
	METHOD AppendCircle
	VAR_IN_OUT
		(* Start position of the circle. *)
 {attribute 'GUID' := '684B7065-E3A9-208A-688F-6768C580A855'}
				startPos : PositionXYC;
		(* End position of the circle. *)
 {attribute 'GUID' := '684B7065-E3A9-208A-688F-6768C580A855'}
				endPos : PositionXYC;
		(* Center of the circle. *)
 {attribute 'GUID' := 'ED71C9D8-8E4B-28CC-7DA0-249C4B114DE7'}
				center : PositionXY;
	END_VAR
	VAR_INPUT
		(* Set whether the circle runs clockwise or counter-clockwise. *)
		clockwise : BOOL;
	END_VAR
END_METHOD


	(* Appends a smooth transition from the end of this path
				      to the start of the other path, locking further changes of this path. *)
	METHOD EndAtPath
	VAR_IN_OUT
		(* The other path. *)
 {attribute 'GUID' := '7FCF97B8-20CD-2CA3-6B3F-E4AF29A0B8D7'}
				path : PathXYC;
	END_VAR
END_METHOD


	(* Appends a smooth transition from the start of this path
				      to the end of the other path, locking further changes of the other path. *)
	METHOD StartFromPath
	VAR_IN_OUT
		(* The other path. *)
 {attribute 'GUID' := '7FCF97B8-20CD-2CA3-6B3F-E4AF29A0B8D7'}
				path : PathXYC;
	END_VAR
END_METHOD


	(* Connect start and end position.
				      A smooth transition is added as long as start and end positin are not identical.
				      This operation finalizes this path definition and locks it against further modifications. *)
	METHOD CloseLoop
END_METHOD


	(* Empty all current path definitions and reset the path back to an empty state. *)
	METHOD Clear
END_METHOD


	(* Get the start position of the path. *)
	METHOD GetStartPosition
	VAR_IN_OUT
		(* The current start position of the path. *)
 {attribute 'GUID' := '684B7065-E3A9-208A-688F-6768C580A855'}
				startPosition : PositionXYC;
	END_VAR
END_METHOD


	(* Get the end position of the segment. *)
	METHOD GetEndPosition
	VAR_IN_OUT
		(* The current end position of the segment. *)
 {attribute 'GUID' := '684B7065-E3A9-208A-688F-6768C580A855'}
				endPosition : PositionXYC;
	END_VAR
END_METHOD


	(* Get a position on the path at a specific arclength value. *)
	METHOD GetPositionAt
	VAR_INPUT
		(* Arc length value where the position is evaluated. *)
		arcLength : LREAL;
	END_VAR
	VAR_IN_OUT
		(* The position at the specified arc parameter. *)
 {attribute 'GUID' := '684B7065-E3A9-208A-688F-6768C580A855'}
				position : PositionXYC;
	END_VAR
END_METHOD


	(* Get the dynamic information when moving along a path
				    with specific arclength value and dynamic changes. *)
	METHOD GetStateAt
	VAR_INPUT
		(* Arc length value where the position is evaluated. *)
		arcLength : LREAL;
		(* Velocity of the arc length parameter. *)
		arcVelocity : LREAL;
		(* Acceleration of the arc length parameter. *)
		arcAcceleration : LREAL;
	END_VAR
	VAR_IN_OUT
		(* The position at the specified arc parameter. *)
 {attribute 'GUID' := '684B7065-E3A9-208A-688F-6768C580A855'}
				position : PositionXYC;
		(* The velocity at the specified dynamic state. *)
 {attribute 'GUID' := 'DC91344B-7822-2D7D-63B8-AA132CC40F5B'}
				velocity : TangentXYC;
		(* The acceleration at the specified dynamic state. *)
 {attribute 'GUID' := 'DC91344B-7822-2D7D-63B8-AA132CC40F5B'}
				acceleration : TangentXYC;
	END_VAR
END_METHOD

END_FUNCTION_BLOCK

// POUs/Shapes/Geometry3D/Container3D

	{attribute 'c++_compatible'}
	{attribute 'external_name' := 'Container3D_GUID_EBD2FAF5_1D6B_25BF_553D_FB39314AE929'}
	{attribute 'TcIecLibraryType'}
	{attribute 'no_explicit_call' :='do not call this POU directly'}
	{attribute 'no_assign'}
	FUNCTION_BLOCK Container3D EXTENDS Geometry3D


	(* Internal method *)
	METHOD FB_init : BOOL
	VAR_INPUT
		(*  if TRUE, the retain variables are initialized (warm start / cold start) *)
		bInitRetains : BOOL;
		(*  if TRUE, the instance afterwards gets moved into the copy code (online change) *)
		bInCopyCode : BOOL;
	END_VAR
END_METHOD


	(* Internal method *)
	{attribute 'hide'}
	METHOD FB_exit : BOOL
	VAR_INPUT
		(*  if TRUE, the exit method is called for exiting an instance that is copied afterwards (online change). *)
		bInCopyCode : BOOL;
	END_VAR
END_METHOD


	(* Add a geometry to the container. *)
	METHOD AddElement : UDINT
	VAR_IN_OUT
		(* The geometry to add. *)
 {attribute 'GUID' := '6A3FD3E0-12B5-2252-6001-2E5EA509DA49'}
				geometry : Geometry3D;
	END_VAR
END_METHOD


	(* Remove a specified geometry from the container. *)
	METHOD RemoveElement
	VAR_INPUT
		(* Identifier of the geometry to remove. *)
		id : UDINT;
	END_VAR
END_METHOD


	(* Remove all geometries from container. *)
	METHOD Clear
END_METHOD


	(* Get the number of geometry elements in container. *)
	METHOD GetCount : UDINT
END_METHOD

END_FUNCTION_BLOCK

// POUs/Shapes/Geometry3D/Extrude3D

	{attribute 'c++_compatible'}
	{attribute 'external_name' := 'Extrude3D_GUID_A12A3BFA_DDAD_26F3_516B_C2FE90166BB2'}
	{attribute 'TcIecLibraryType'}
	{attribute 'no_explicit_call' :='do not call this POU directly'}
	{attribute 'no_assign'}
	FUNCTION_BLOCK Extrude3D EXTENDS Geometry3D


	(* Internal method *)
	METHOD FB_init : BOOL
	VAR_INPUT
		(*  if TRUE, the retain variables are initialized (warm start / cold start) *)
		bInitRetains : BOOL;
		(*  if TRUE, the instance afterwards gets moved into the copy code (online change) *)
		bInCopyCode : BOOL;
	END_VAR
END_METHOD


	(* Internal method *)
	{attribute 'hide'}
	METHOD FB_exit : BOOL
	VAR_INPUT
		(*  if TRUE, the exit method is called for exiting an instance that is copied afterwards (online change). *)
		bInCopyCode : BOOL;
	END_VAR
END_METHOD


	(* Define the extrude geometry with a path and a array of xy-points *)
	METHOD DefineByPath : BOOL
	VAR_IN_OUT
		(* Cross section values *)
 {attribute 'GUID' := 'ED71C9D8-8E4B-28CC-7DA0-249C4B114DE7'}
				PointerToCrossSection : POINTER TO PositionXY;
	END_VAR
	VAR_INPUT
		(* Number of cross section points *)
		NumberOfCrossSectionPoints : UDINT;
	END_VAR
	VAR_IN_OUT
		(* The path *)
 {attribute 'GUID' := '59C0DC94-4833-2811-5F1B-49E2178993C5'}
				Path : PathXYZ;
	END_VAR
	VAR_INPUT
		(* Number of path points *)
		NumberOfPathPoints : UDINT;
	END_VAR
END_METHOD

END_FUNCTION_BLOCK

// POUs/Paths/Components/PathXYZ

	{attribute 'c++_compatible'}
	{attribute 'external_name' := 'PathXYZ_GUID_59C0DC94_4833_2811_5F1B_49E2178993C5'}
	{attribute 'TcIecLibraryType'}
	{attribute 'no_explicit_call' :='do not call this POU directly'}
	{attribute 'no_assign'}
	(* A path in the xy-plane with an additional orientation at every path position. *)
	FUNCTION_BLOCK PathXYZ EXTENDS IPlcPath3D


	(* Internal method *)
	{attribute 'hide'}
	METHOD FB_init : BOOL
	VAR_INPUT
		(*  if TRUE, the retain variables are initialized (warm start / cold start) *)
		bInitRetains : BOOL;
		(*  if TRUE, the instance afterwards gets moved into the copy code (online change) *)
		bInCopyCode : BOOL;
	END_VAR
END_METHOD


	(* Internal method *)
	{attribute 'hide'}
	METHOD FB_exit : BOOL
	VAR_INPUT
		(*  if TRUE, the exit method is called for exiting an instance that is copied afterwards (online change). *)
		bInCopyCode : BOOL;
	END_VAR
END_METHOD


	(* Append a smooth transition from the current end of the path
				    to the specified position. *)
	METHOD AppendPosition
	VAR_IN_OUT
		(* The position to append. *)
 {attribute 'GUID' := '513B7ECA-E1D5-262C-5763-788E1FD4F5AD'}
				position : Position3D;
	END_VAR
END_METHOD


	(* Append a smooth transition from the current end of the path
				    to the specified position. *)
	METHOD AppendPositionXYZ
	VAR_INPUT
		(* x-component of the position to append. *)
		x : LREAL;
		(* y-component of the position to append. *)
		y : LREAL;
		(* z-component of the position to append. *)
		c : LREAL;
	END_VAR
END_METHOD


	(* Append a line to this path. *)
	METHOD AppendLine
	VAR_IN_OUT
		(* Start position of the line. *)
 {attribute 'GUID' := '513B7ECA-E1D5-262C-5763-788E1FD4F5AD'}
				startPos : Position3D;
		(* End position of the line. *)
 {attribute 'GUID' := '513B7ECA-E1D5-262C-5763-788E1FD4F5AD'}
				endPos : Position3D;
	END_VAR
END_METHOD


	(* Append a smooth transition from the current end of the path
				    to the specified position. *)
	METHOD AppendLineXYZ
	VAR_INPUT
		(* x-component of the start position. *)
		x0 : LREAL;
		(* y-component of the start position. *)
		y0 : LREAL;
		(* z-component of the start position. *)
		z0 : LREAL;
		(* x-component of the end position. *)
		x1 : LREAL;
		(* y-component of the end position. *)
		y1 : LREAL;
		(* z-component of the end position. *)
		z1 : LREAL;
	END_VAR
END_METHOD


	(* Append a circle to this path. *)
	METHOD AppendCircle
	VAR_IN_OUT
		(* Start position of the circle. *)
 {attribute 'GUID' := '513B7ECA-E1D5-262C-5763-788E1FD4F5AD'}
				startPos : Position3D;
		(* End position of the circle. *)
 {attribute 'GUID' := '513B7ECA-E1D5-262C-5763-788E1FD4F5AD'}
				endPos : Position3D;
		(* Center of the circle. *)
 {attribute 'GUID' := 'ED71C9D8-8E4B-28CC-7DA0-249C4B114DE7'}
				center : PositionXY;
	END_VAR
	VAR_INPUT
		(* Set whether the circle runs clockwise or counter-clockwise. *)
		clockwise : BOOL;
	END_VAR
END_METHOD


	(* Append a smooth transition from the current end of the path
				    to the specified position with tangent. *)
	METHOD AppendPositionTangent
	VAR_IN_OUT
		(* The position to append. *)
 {attribute 'GUID' := '513B7ECA-E1D5-262C-5763-788E1FD4F5AD'}
				position : Position3D;
		(* The tangent to append *)
 {attribute 'GUID' := '8E451EF0-1EF7-2C22-40FE-C3C408FD9C3F'}
				tangent : Tangent3D;
	END_VAR
END_METHOD


	(* Get the start position of the path. *)
	METHOD GetStartPosition
	VAR_IN_OUT
		(* The current start position of the path. *)
 {attribute 'GUID' := '513B7ECA-E1D5-262C-5763-788E1FD4F5AD'}
				startPosition : Position3D;
	END_VAR
END_METHOD


	(* Get the end position of the segment. *)
	METHOD GetEndPosition
	VAR_IN_OUT
		(* The current end position of the segment. *)
 {attribute 'GUID' := '513B7ECA-E1D5-262C-5763-788E1FD4F5AD'}
				endPosition : Position3D;
	END_VAR
END_METHOD


	(* Get a position on the path at a specific arclength value. *)
	METHOD GetPositionAt
	VAR_INPUT
		(* Arc length value where the position is evaluated. *)
		arcLength : LREAL;
	END_VAR
	VAR_IN_OUT
		(* The position at the specified arc parameter. *)
 {attribute 'GUID' := '513B7ECA-E1D5-262C-5763-788E1FD4F5AD'}
				position : Position3D;
	END_VAR
END_METHOD


	(* Get the dynamic information when moving along a path
				    with specific arclength value and dynamic changes. *)
	METHOD GetStateAt
	VAR_INPUT
		(* Arc length value where the position is evaluated. *)
		arcLength : LREAL;
		(* Velocity of the arc length parameter. *)
		arcVelocity : LREAL;
		(* Acceleration of the arc length parameter. *)
		arcAcceleration : LREAL;
	END_VAR
	VAR_IN_OUT
		(* The position at the specified arc parameter. *)
 {attribute 'GUID' := '513B7ECA-E1D5-262C-5763-788E1FD4F5AD'}
				position : Position3D;
		(* The velocity at the specified dynamic state. *)
 {attribute 'GUID' := '8E451EF0-1EF7-2C22-40FE-C3C408FD9C3F'}
				velocity : Tangent3D;
		(* The acceleration at the specified dynamic state. *)
 {attribute 'GUID' := '8E451EF0-1EF7-2C22-40FE-C3C408FD9C3F'}
				acceleration : Tangent3D;
	END_VAR
END_METHOD

END_FUNCTION_BLOCK

// POUs/Paths/Components/PathXY

	{attribute 'c++_compatible'}
	{attribute 'external_name' := 'PathXY_GUID_BE2746EF_23B4_26FF_7005_FB1D2BCFB3FC'}
	{attribute 'TcIecLibraryType'}
	{attribute 'no_explicit_call' :='do not call this POU directly'}
	{attribute 'no_assign'}
	(* A path in the xy-plane. *)
	FUNCTION_BLOCK PathXY EXTENDS IPlcPath2D


	(* Internal method *)
	{attribute 'hide'}
	METHOD FB_init : BOOL
	VAR_INPUT
		(*  if TRUE, the retain variables are initialized (warm start / cold start) *)
		bInitRetains : BOOL;
		(*  if TRUE, the instance afterwards gets moved into the copy code (online change) *)
		bInCopyCode : BOOL;
	END_VAR
END_METHOD


	(* Internal method *)
	{attribute 'hide'}
	METHOD FB_exit : BOOL
	VAR_INPUT
		(*  if TRUE, the exit method is called for exiting an instance that is copied afterwards (online change). *)
		bInCopyCode : BOOL;
	END_VAR
END_METHOD


	(* Append a smooth transition from the current end of the path
				    to the specified position. *)
	METHOD AppendPosition
	VAR_IN_OUT
		(* The position to append. *)
 {attribute 'GUID' := 'ED71C9D8-8E4B-28CC-7DA0-249C4B114DE7'}
				position : PositionXY;
	END_VAR
END_METHOD


	(* Append a smooth transition from the current end of the path
				    to the specified position. *)
	METHOD AppendPositionXY
	VAR_INPUT
		(* x-component of the position to append. *)
		x : LREAL;
		(* y-component of the position to append. *)
		y : LREAL;
	END_VAR
END_METHOD


	(* Append a line to this path. *)
	METHOD AppendLine
	VAR_IN_OUT
		(* Start position of the line. *)
 {attribute 'GUID' := 'ED71C9D8-8E4B-28CC-7DA0-249C4B114DE7'}
				startPos : PositionXY;
		(* End position of the line. *)
 {attribute 'GUID' := 'ED71C9D8-8E4B-28CC-7DA0-249C4B114DE7'}
				endPos : PositionXY;
	END_VAR
END_METHOD


	(* Append a circle to this path. *)
	METHOD AppendCircle
	VAR_IN_OUT
		(* Start position of the circle. *)
 {attribute 'GUID' := 'ED71C9D8-8E4B-28CC-7DA0-249C4B114DE7'}
				startPos : PositionXY;
		(* End position of the circle. *)
 {attribute 'GUID' := 'ED71C9D8-8E4B-28CC-7DA0-249C4B114DE7'}
				endPos : PositionXY;
		(* Center of the circle. *)
 {attribute 'GUID' := 'ED71C9D8-8E4B-28CC-7DA0-249C4B114DE7'}
				center : PositionXY;
	END_VAR
	VAR_INPUT
		(* Set whether the circle runs clockwise or counter-clockwise. *)
		clockwise : BOOL;
	END_VAR
END_METHOD


	(* Get the start position of the path. *)
	METHOD GetStartPosition
	VAR_IN_OUT
		(* The current start position of the path. *)
 {attribute 'GUID' := 'ED71C9D8-8E4B-28CC-7DA0-249C4B114DE7'}
				startPosition : PositionXY;
	END_VAR
END_METHOD


	(* Get the end position of the segment. *)
	METHOD GetEndPosition
	VAR_IN_OUT
		(* The current end position of the segment. *)
 {attribute 'GUID' := 'ED71C9D8-8E4B-28CC-7DA0-249C4B114DE7'}
				endPosition : PositionXY;
	END_VAR
END_METHOD


	(* Get a position on the path at a specific arclength value. *)
	METHOD GetPositionAt
	VAR_INPUT
		(* Arc length value where the position is evaluated. *)
		arcLength : LREAL;
	END_VAR
	VAR_IN_OUT
		(* The position at the specified arc parameter. *)
 {attribute 'GUID' := 'ED71C9D8-8E4B-28CC-7DA0-249C4B114DE7'}
				position : PositionXY;
	END_VAR
END_METHOD


	(* Get the dynamic information when moving along a path
				    with specific arclength value and dynamic changes. *)
	METHOD GetStateAt
	VAR_INPUT
		(* Arc length value where the position is evaluated. *)
		arcLength : LREAL;
		(* Velocity of the arc length parameter. *)
		arcVelocity : LREAL;
		(* Acceleration of the arc length parameter. *)
		arcAcceleration : LREAL;
	END_VAR
	VAR_IN_OUT
		(* The position at the specified arc parameter. *)
 {attribute 'GUID' := 'ED71C9D8-8E4B-28CC-7DA0-249C4B114DE7'}
				position : PositionXY;
		(* The velocity at the specified dynamic state. *)
 {attribute 'GUID' := '5D3BC02D-EA16-22EA-7ADA-76A9B505DC98'}
				velocity : TangentXY;
		(* The acceleration at the specified dynamic state. *)
 {attribute 'GUID' := '5D3BC02D-EA16-22EA-7ADA-76A9B505DC98'}
				acceleration : TangentXY;
	END_VAR
END_METHOD

END_FUNCTION_BLOCK

// POUs/Shapes/Geometry2D/1D/Line2D

	{attribute 'c++_compatible'}
	{attribute 'external_name' := 'Line2D_GUID_AAAE24FC_F23F_2E46_7C02_8AD42345D7DE'}
	{attribute 'TcIecLibraryType'}
	{attribute 'no_explicit_call' :='do not call this POU directly'}
	{attribute 'no_assign'}
	(* 2D Geometry Line *)
	FUNCTION_BLOCK Line2D EXTENDS Geometry2D


	(* Internal method *)
	METHOD FB_init : BOOL
	VAR_INPUT
		(*  if TRUE, the retain variables are initialized (warm start / cold start) *)
		bInitRetains : BOOL;
		(*  if TRUE, the instance afterwards gets moved into the copy code (online change) *)
		bInCopyCode : BOOL;
	END_VAR
END_METHOD


	(* Internal method *)
	{attribute 'hide'}
	METHOD FB_exit : BOOL
	VAR_INPUT
		(*  if TRUE, the exit method is called for exiting an instance that is copied afterwards (online change). *)
		bInCopyCode : BOOL;
	END_VAR
END_METHOD


	(* Define a line by two positions. *)
	METHOD DefineByPositions
	VAR_IN_OUT
		(* 1st position on the line to define. *)
 {attribute 'GUID' := 'ED71C9D8-8E4B-28CC-7DA0-249C4B114DE7'}
				position0 : PositionXY;
		(* 2nd position on the line to define. *)
 {attribute 'GUID' := 'ED71C9D8-8E4B-28CC-7DA0-249C4B114DE7'}
				position1 : PositionXY;
	END_VAR
END_METHOD


	(* Define a line by a position on the line and its direction. *)
	METHOD DefineByDirection
	VAR_IN_OUT
		(* Position on the line *)
 {attribute 'GUID' := 'ED71C9D8-8E4B-28CC-7DA0-249C4B114DE7'}
				position : PositionXY;
		(* Direction of the line *)
 {attribute 'GUID' := '5D3BC02D-EA16-22EA-7ADA-76A9B505DC98'}
				direction : TangentXY;
	END_VAR
END_METHOD


	(* Set the direction of the line. *)
	METHOD SetDirection
	VAR_IN_OUT
		(* The direction to set. *)
 {attribute 'GUID' := '5D3BC02D-EA16-22EA-7ADA-76A9B505DC98'}
				direction : TangentXY;
	END_VAR
END_METHOD


	(* Get the direction of the line. *)
	METHOD GetDirection
	VAR_IN_OUT
		(* The current direction of the line. *)
 {attribute 'GUID' := '5D3BC02D-EA16-22EA-7ADA-76A9B505DC98'}
				direction : TangentXY;
	END_VAR
END_METHOD


	(* Get a position on the line at a specific arclength value. *)
	METHOD GetPositionAt
	VAR_INPUT
		(* Arc length value where the position is evaluated. *)
		arcLength : LREAL;
	END_VAR
	VAR_IN_OUT
		(* The position at the specified arc parameter. *)
 {attribute 'GUID' := '684B7065-E3A9-208A-688F-6768C580A855'}
				position : PositionXYC;
	END_VAR
END_METHOD

END_FUNCTION_BLOCK

// POUs/Shapes/Geometry2D/1D/Segment2D

	{attribute 'c++_compatible'}
	{attribute 'external_name' := 'Segment2D_GUID_CB5FC4F9_F3B9_2658_7F54_FF048B094404'}
	{attribute 'TcIecLibraryType'}
	{attribute 'no_explicit_call' :='do not call this POU directly'}
	{attribute 'no_assign'}
	FUNCTION_BLOCK Segment2D EXTENDS Geometry2D


	(* Internal method *)
	METHOD FB_init : BOOL
	VAR_INPUT
		(*  if TRUE, the retain variables are initialized (warm start / cold start) *)
		bInitRetains : BOOL;
		(*  if TRUE, the instance afterwards gets moved into the copy code (online change) *)
		bInCopyCode : BOOL;
	END_VAR
END_METHOD


	(* Internal method *)
	{attribute 'hide'}
	METHOD FB_exit : BOOL
	VAR_INPUT
		(*  if TRUE, the exit method is called for exiting an instance that is copied afterwards (online change). *)
		bInCopyCode : BOOL;
	END_VAR
END_METHOD


	(* Set the start position of the segment. *)
	METHOD SetStartPosition
	VAR_IN_OUT
		(* Start position of the segment to set. *)
 {attribute 'GUID' := 'ED71C9D8-8E4B-28CC-7DA0-249C4B114DE7'}
				startPos : PositionXY;
	END_VAR
END_METHOD


	(* Set the start position of the segment. *)
	METHOD SetStartPositionXY
	VAR_INPUT
		(* x-component of the start position. *)
		x : LREAL;
		(* y-component of the start position. *)
		y : LREAL;
	END_VAR
END_METHOD


	(* Set the end position of the segment. *)
	METHOD SetEndPosition
	VAR_IN_OUT
		(* End position of the segment to set. *)
 {attribute 'GUID' := 'ED71C9D8-8E4B-28CC-7DA0-249C4B114DE7'}
				endPos : PositionXY;
	END_VAR
END_METHOD


	(* Set the end position of the segment. *)
	METHOD SetEndPositionXY
	VAR_INPUT
		(* x-component of the end position. *)
		x : LREAL;
		(* y-component of the end position. *)
		y : LREAL;
	END_VAR
END_METHOD


	(* Get the x-component of the segment length in respect to the root coordinate system. *)
	METHOD Get_dX : LREAL
END_METHOD


	(* Get the y-component of the segment length in respect to the root coordinate system. *)
	METHOD Get_dY : LREAL
END_METHOD


	(* Get the length of the segment. *)
	METHOD GetLength : LREAL
END_METHOD


	(* Get the start position of the segment. *)
	METHOD GetStartPosition
	VAR_IN_OUT
		(* The current start position of the segment. *)
 {attribute 'GUID' := 'ED71C9D8-8E4B-28CC-7DA0-249C4B114DE7'}
				startPosition : PositionXY;
	END_VAR
END_METHOD


	(* Get the end position of the segment. *)
	METHOD GetEndPosition
	VAR_IN_OUT
		(* The current end position of the segment. *)
 {attribute 'GUID' := 'ED71C9D8-8E4B-28CC-7DA0-249C4B114DE7'}
				endPosition : PositionXY;
	END_VAR
END_METHOD


	(* Get the direction of the segment. *)
	METHOD GetDirection
	VAR_IN_OUT
		(* The current direction of the segment. *)
 {attribute 'GUID' := '5D3BC02D-EA16-22EA-7ADA-76A9B505DC98'}
				direction : TangentXY;
	END_VAR
END_METHOD


	(* Get a position on the segment at a specific arclength value. *)
	METHOD GetPositionAt
	VAR_INPUT
		(* Arc length value where the position is evaluated. *)
		arcLength : LREAL;
	END_VAR
	VAR_IN_OUT
		(* The position at the specified arc parameter. *)
 {attribute 'GUID' := '684B7065-E3A9-208A-688F-6768C580A855'}
				position : PositionXYC;
	END_VAR
END_METHOD

END_FUNCTION_BLOCK

// POUs/Shapes/Geometry2D/1D/Circle2D

	{attribute 'c++_compatible'}
	{attribute 'external_name' := 'Circle2D_GUID_9C18178A_FF25_2591_4D8E_DD34ADA001A5'}
	{attribute 'TcIecLibraryType'}
	{attribute 'no_explicit_call' :='do not call this POU directly'}
	{attribute 'no_assign'}
	FUNCTION_BLOCK Circle2D EXTENDS Geometry2D


	(* Internal method *)
	METHOD FB_init : BOOL
	VAR_INPUT
		(*  if TRUE, the retain variables are initialized (warm start / cold start) *)
		bInitRetains : BOOL;
		(*  if TRUE, the instance afterwards gets moved into the copy code (online change) *)
		bInCopyCode : BOOL;
	END_VAR
END_METHOD


	(* Internal method *)
	{attribute 'hide'}
	METHOD FB_exit : BOOL
	VAR_INPUT
		(*  if TRUE, the exit method is called for exiting an instance that is copied afterwards (online change). *)
		bInCopyCode : BOOL;
	END_VAR
END_METHOD


	(* Get the length of the circle. *)
	METHOD GetLength : LREAL
END_METHOD


	(* Get a position on the circle at a specific arclength value. *)
	METHOD GetPositionAt
	VAR_INPUT
		(* Arc length value where the position is evaluated. *)
		arcLength : LREAL;
	END_VAR
	VAR_IN_OUT
		(* The position at the specified arc parameter. *)
 {attribute 'GUID' := '684B7065-E3A9-208A-688F-6768C580A855'}
				position : PositionXYC;
	END_VAR
END_METHOD


	PROPERTY radius : LREAL
GET
END_GET
SET
END_SET
END_PROPERTY

END_FUNCTION_BLOCK

// POUs/Shapes/Geometry2D/2D/Disc2D

	{attribute 'c++_compatible'}
	{attribute 'external_name' := 'Disc2D_GUID_61EF6B64_61FE_2C67_55CC_5655A9B10489'}
	{attribute 'TcIecLibraryType'}
	{attribute 'no_explicit_call' :='do not call this POU directly'}
	{attribute 'no_assign'}
	FUNCTION_BLOCK Disc2D EXTENDS Geometry2D


	(* Internal method *)
	METHOD FB_init : BOOL
	VAR_INPUT
		(*  if TRUE, the retain variables are initialized (warm start / cold start) *)
		bInitRetains : BOOL;
		(*  if TRUE, the instance afterwards gets moved into the copy code (online change) *)
		bInCopyCode : BOOL;
	END_VAR
END_METHOD


	(* Internal method *)
	{attribute 'hide'}
	METHOD FB_exit : BOOL
	VAR_INPUT
		(*  if TRUE, the exit method is called for exiting an instance that is copied afterwards (online change). *)
		bInCopyCode : BOOL;
	END_VAR
END_METHOD


	(* Get the area of the disc. *)
	METHOD GetArea : LREAL
END_METHOD


	PROPERTY radius : LREAL
GET
END_GET
SET
END_SET
END_PROPERTY

END_FUNCTION_BLOCK

// POUs/Shapes/Geometry2D/2D/Rectangle2D

	{attribute 'c++_compatible'}
	{attribute 'external_name' := 'Rectangle2D_GUID_4FCD58F9_E59B_202F_4E14_ED5CB4562B9B'}
	{attribute 'TcIecLibraryType'}
	{attribute 'no_explicit_call' :='do not call this POU directly'}
	{attribute 'no_assign'}
	FUNCTION_BLOCK Rectangle2D EXTENDS Geometry2D


	(* Internal method *)
	METHOD FB_init : BOOL
	VAR_INPUT
		(*  if TRUE, the retain variables are initialized (warm start / cold start) *)
		bInitRetains : BOOL;
		(*  if TRUE, the instance afterwards gets moved into the copy code (online change) *)
		bInCopyCode : BOOL;
	END_VAR
END_METHOD


	(* Internal method *)
	{attribute 'hide'}
	METHOD FB_exit : BOOL
	VAR_INPUT
		(*  if TRUE, the exit method is called for exiting an instance that is copied afterwards (online change). *)
		bInCopyCode : BOOL;
	END_VAR
END_METHOD


	(* Set the dimensions of the rectangle. *)
	METHOD SetDimensions
	VAR_INPUT
		(* The width of the rectangle to set. *)
		width : LREAL;
		(* The height of the rectangle to set. *)
		height : LREAL;
	END_VAR
END_METHOD


	(* Get the area of the rectangle. *)
	METHOD GetArea : LREAL
END_METHOD


	PROPERTY width : LREAL
GET
END_GET
SET
END_SET
END_PROPERTY


	PROPERTY height : LREAL
GET
END_GET
SET
END_SET
END_PROPERTY

END_FUNCTION_BLOCK

// POUs/Shapes/Geometry2D/Functions/CheckCollision2D

	{attribute 'TcIecLibraryType'}
	{attribute 'external_name' := 'CheckCollision2D_GUID_F17EC77E_7F62_2BD1_4356_756430091B1F'}
	(* Check if two geometries are currently colliding. *)
	FUNCTION CheckCollision2D : BOOL
	VAR_IN_OUT
		geometry0	:	IPlcGeometry2D;	(* 1st input geometry to check for collision. *)
		geometry1	:	IPlcGeometry2D;	(* 2nd input geometry to check of collision. *)
	END_VAR

END_FUNCTION

// POUs/Shapes/Geometry2D/Functions/GetDistance2D

	{attribute 'TcIecLibraryType'}
	{attribute 'external_name' := 'GetDistance2D_GUID_CEB1BC86_BE19_2144_771A_7B4585B2C683'}
	(* Get the distance between two geometries. *)
	FUNCTION GetDistance2D : LREAL
	VAR_IN_OUT
		geometry0	:	IPlcGeometry2D;	(* 1st input geometry to calculate the distance of. *)
		geometry1	:	IPlcGeometry2D;	(* 2nd input geometry to calculate the distance of. *)
	END_VAR

END_FUNCTION

// POUs/Shapes/Geometry2D/Functions/GetLinkingLine2D

	{attribute 'TcIecLibraryType'}
	{attribute 'external_name' := 'GetLinkingLine2D_GUID_885ABCB9_CCEF_2F29_5364_14DECC9E69D5'}
	(* Get the shortest path between two geometries. *)
	FUNCTION GetLinkingLine2D : BOOL
	VAR_IN_OUT
		geometry0	:	IPlcGeometry2D;	(* 1st input geometry to calculate the linking line for. *)
		geometry1	:	IPlcGeometry2D;	(* 2nd input geometry to calculate the linking line for. *)
		linkingLine	:	Segment2D;	(* Return the resulting linking line. *)
	END_VAR

END_FUNCTION

// POUs/Shapes/Geometry3D/1D/Line3D

	{attribute 'c++_compatible'}
	{attribute 'external_name' := 'Line3D_GUID_A7105F73_A0CA_26BA_559B_EF5477D3CFC5'}
	{attribute 'TcIecLibraryType'}
	{attribute 'no_explicit_call' :='do not call this POU directly'}
	{attribute 'no_assign'}
	(* 3D Geometry Line *)
	FUNCTION_BLOCK Line3D EXTENDS Geometry3D


	(* Internal method *)
	METHOD FB_init : BOOL
	VAR_INPUT
		(*  if TRUE, the retain variables are initialized (warm start / cold start) *)
		bInitRetains : BOOL;
		(*  if TRUE, the instance afterwards gets moved into the copy code (online change) *)
		bInCopyCode : BOOL;
	END_VAR
END_METHOD


	(* Internal method *)
	{attribute 'hide'}
	METHOD FB_exit : BOOL
	VAR_INPUT
		(*  if TRUE, the exit method is called for exiting an instance that is copied afterwards (online change). *)
		bInCopyCode : BOOL;
	END_VAR
END_METHOD


	(* Define a line by two positions. *)
	METHOD DefineByPositions
	VAR_IN_OUT
		(* 1st position on the line to define. *)
 {attribute 'GUID' := '513B7ECA-E1D5-262C-5763-788E1FD4F5AD'}
				position0 : Position3D;
		(* 2nd position on the line to define. *)
 {attribute 'GUID' := '513B7ECA-E1D5-262C-5763-788E1FD4F5AD'}
				position1 : Position3D;
	END_VAR
END_METHOD


	(* Define a line by a position on the line and its direction. *)
	METHOD DefineByDirection
	VAR_IN_OUT
		(* Position on the line. *)
 {attribute 'GUID' := '513B7ECA-E1D5-262C-5763-788E1FD4F5AD'}
				position : Position3D;
		(* Direction of the line. *)
 {attribute 'GUID' := '8E451EF0-1EF7-2C22-40FE-C3C408FD9C3F'}
				direction : Tangent3D;
	END_VAR
END_METHOD


	(* Set the direction of the line. *)
	METHOD SetDirection
	VAR_IN_OUT
		(* The direction to set. *)
 {attribute 'GUID' := '8E451EF0-1EF7-2C22-40FE-C3C408FD9C3F'}
				direction : Tangent3D;
	END_VAR
END_METHOD


	(* Get the direction of the line. *)
	METHOD GetDirection
	VAR_IN_OUT
		(* The current direction of the line. *)
 {attribute 'GUID' := '8E451EF0-1EF7-2C22-40FE-C3C408FD9C3F'}
				direction : Tangent3D;
	END_VAR
END_METHOD


	(* Get a position on the line at a specific arclength value. *)
	METHOD GetPositionAt
	VAR_INPUT
		(* Arc length value where the position is evaluated. *)
		arcLength : LREAL;
	END_VAR
	VAR_IN_OUT
		(* The position at the specified arc parameter. *)
 {attribute 'GUID' := '71570C9B-708B-2C60-4B94-668F28922D38'}
				position : PositionSE3;
	END_VAR
END_METHOD

END_FUNCTION_BLOCK

// POUs/Shapes/Geometry3D/1D/Segment3D

	{attribute 'c++_compatible'}
	{attribute 'external_name' := 'Segment3D_GUID_9AC14DE1_1F36_219E_4DB2_90E090430F95'}
	{attribute 'TcIecLibraryType'}
	{attribute 'no_explicit_call' :='do not call this POU directly'}
	{attribute 'no_assign'}
	FUNCTION_BLOCK Segment3D EXTENDS Geometry3D


	(* Internal method *)
	METHOD FB_init : BOOL
	VAR_INPUT
		(*  if TRUE, the retain variables are initialized (warm start / cold start) *)
		bInitRetains : BOOL;
		(*  if TRUE, the instance afterwards gets moved into the copy code (online change) *)
		bInCopyCode : BOOL;
	END_VAR
END_METHOD


	(* Internal method *)
	{attribute 'hide'}
	METHOD FB_exit : BOOL
	VAR_INPUT
		(*  if TRUE, the exit method is called for exiting an instance that is copied afterwards (online change). *)
		bInCopyCode : BOOL;
	END_VAR
END_METHOD


	(* Set the start position of the segment. *)
	METHOD SetStartPosition
	VAR_IN_OUT
		(* Start position of the segment to set. *)
 {attribute 'GUID' := '513B7ECA-E1D5-262C-5763-788E1FD4F5AD'}
				startPos : Position3D;
	END_VAR
END_METHOD


	(* Set the start position of the segment. *)
	METHOD SetStartPositionXYZ
	VAR_INPUT
		(* x-component of the start position. *)
		x : LREAL;
		(* y-component of the start position. *)
		y : LREAL;
		(* z-component of the start position. *)
		z : LREAL;
	END_VAR
END_METHOD


	(* Set the end position of the segment. *)
	METHOD SetEndPosition
	VAR_IN_OUT
		(* End position of the segment to set. *)
 {attribute 'GUID' := '513B7ECA-E1D5-262C-5763-788E1FD4F5AD'}
				endPos : Position3D;
	END_VAR
END_METHOD


	(* Set the end position of the segment. *)
	METHOD SetEndPositionXYZ
	VAR_INPUT
		(* x-component of the end position. *)
		x : LREAL;
		(* y-component of the end position. *)
		y : LREAL;
		(* z-component of the end position. *)
		z : LREAL;
	END_VAR
END_METHOD


	(* Get the x-component of the segment length in respect to the root coordinate system. *)
	METHOD Get_dX : LREAL
END_METHOD


	(* Get the y-component of the segment length in respect to the root coordinate system. *)
	METHOD Get_dY : LREAL
END_METHOD


	(* Get the z-component of the segment length in respect to the root coordinate system. *)
	METHOD Get_dZ : LREAL
END_METHOD


	(* Get the length of the segment. *)
	METHOD GetLength : LREAL
END_METHOD


	(* Get the start position of the segment. *)
	METHOD GetStartPosition
	VAR_IN_OUT
		(* The current start position of the segment. *)
 {attribute 'GUID' := '513B7ECA-E1D5-262C-5763-788E1FD4F5AD'}
				startPosition : Position3D;
	END_VAR
END_METHOD


	(* Get the end position of the segment. *)
	METHOD GetEndPosition
	VAR_IN_OUT
		(* The current end position of the segment. *)
 {attribute 'GUID' := '513B7ECA-E1D5-262C-5763-788E1FD4F5AD'}
				endPosition : Position3D;
	END_VAR
END_METHOD


	(* Get the direction of the segment. *)
	METHOD GetDirection
	VAR_IN_OUT
		(* The current direction of the segment. *)
 {attribute 'GUID' := '8E451EF0-1EF7-2C22-40FE-C3C408FD9C3F'}
				direction : Tangent3D;
	END_VAR
END_METHOD


	(* Get a position on the segment at a specific arclength value. *)
	METHOD GetPositionAt
	VAR_INPUT
		(* Arc length value where the position is evaluated. *)
		arcLength : LREAL;
	END_VAR
	VAR_IN_OUT
		(* The position at the specified arc parameter. *)
 {attribute 'GUID' := '71570C9B-708B-2C60-4B94-668F28922D38'}
				position : PositionSE3;
	END_VAR
END_METHOD

END_FUNCTION_BLOCK

// POUs/Shapes/Geometry3D/1D/Circle3D

	{attribute 'c++_compatible'}
	{attribute 'external_name' := 'Circle3D_GUID_52779506_23D8_2120_590B_02DAA54ABBF8'}
	{attribute 'TcIecLibraryType'}
	{attribute 'no_explicit_call' :='do not call this POU directly'}
	{attribute 'no_assign'}
	FUNCTION_BLOCK Circle3D EXTENDS Geometry3D


	(* Internal method *)
	METHOD FB_init : BOOL
	VAR_INPUT
		(*  if TRUE, the retain variables are initialized (warm start / cold start) *)
		bInitRetains : BOOL;
		(*  if TRUE, the instance afterwards gets moved into the copy code (online change) *)
		bInCopyCode : BOOL;
	END_VAR
END_METHOD


	(* Internal method *)
	{attribute 'hide'}
	METHOD FB_exit : BOOL
	VAR_INPUT
		(*  if TRUE, the exit method is called for exiting an instance that is copied afterwards (online change). *)
		bInCopyCode : BOOL;
	END_VAR
END_METHOD


	(* Set the normal vector of the circle. *)
	METHOD SetNormal
	VAR_IN_OUT
		(* Normal vector to set. *)
 {attribute 'GUID' := '8E451EF0-1EF7-2C22-40FE-C3C408FD9C3F'}
				normal : Tangent3D;
	END_VAR
END_METHOD


	(* Get the length of the circle. *)
	METHOD GetLength : LREAL
END_METHOD


	(* Get the normal vector of the circle. *)
	METHOD GetNormal
	VAR
		(* The current normal vector of the circle. *)
 {attribute 'GUID' := '8E451EF0-1EF7-2C22-40FE-C3C408FD9C3F'}
				normal : Tangent3D;
	END_VAR
END_METHOD


	(* Get a position on the circle at a specific arclength value. *)
	METHOD GetPositionAt
	VAR_INPUT
		(* Arc length value where the position is evaluated. *)
		arcLength : LREAL;
	END_VAR
	VAR_IN_OUT
		(* The position at the specified arc parameter. *)
 {attribute 'GUID' := '71570C9B-708B-2C60-4B94-668F28922D38'}
				position : PositionSE3;
	END_VAR
END_METHOD


	PROPERTY radius : LREAL
GET
END_GET
SET
END_SET
END_PROPERTY

END_FUNCTION_BLOCK

// POUs/Shapes/Geometry3D/2D/Plane3D

	{attribute 'c++_compatible'}
	{attribute 'external_name' := 'Plane3D_GUID_A3477777_2A55_2AF1_7215_5AAA88F5EEED'}
	{attribute 'TcIecLibraryType'}
	{attribute 'no_explicit_call' :='do not call this POU directly'}
	{attribute 'no_assign'}
	FUNCTION_BLOCK Plane3D EXTENDS Geometry3D


	(* Internal method *)
	METHOD FB_init : BOOL
	VAR_INPUT
		(*  if TRUE, the retain variables are initialized (warm start / cold start) *)
		bInitRetains : BOOL;
		(*  if TRUE, the instance afterwards gets moved into the copy code (online change) *)
		bInCopyCode : BOOL;
	END_VAR
END_METHOD


	(* Internal method *)
	{attribute 'hide'}
	METHOD FB_exit : BOOL
	VAR_INPUT
		(*  if TRUE, the exit method is called for exiting an instance that is copied afterwards (online change). *)
		bInCopyCode : BOOL;
	END_VAR
END_METHOD


	(* Set the normal of the plane. *)
	METHOD SetNormal
	VAR_IN_OUT
		(* The normal vector to set. *)
 {attribute 'GUID' := '8E451EF0-1EF7-2C22-40FE-C3C408FD9C3F'}
				normal : Tangent3D;
	END_VAR
END_METHOD


	(* Get the normal vector of the plane. *)
	METHOD GetNormal
	VAR
		(* The current normal vector of the plane. *)
 {attribute 'GUID' := '8E451EF0-1EF7-2C22-40FE-C3C408FD9C3F'}
				normal : Tangent3D;
	END_VAR
END_METHOD

END_FUNCTION_BLOCK

// POUs/Shapes/Geometry3D/2D/Disc3D

	{attribute 'c++_compatible'}
	{attribute 'external_name' := 'Disc3D_GUID_39F999A8_B8B6_26E5_78BB_0D18E9F380AF'}
	{attribute 'TcIecLibraryType'}
	{attribute 'no_explicit_call' :='do not call this POU directly'}
	{attribute 'no_assign'}
	FUNCTION_BLOCK Disc3D EXTENDS Geometry3D


	(* Internal method *)
	METHOD FB_init : BOOL
	VAR_INPUT
		(*  if TRUE, the retain variables are initialized (warm start / cold start) *)
		bInitRetains : BOOL;
		(*  if TRUE, the instance afterwards gets moved into the copy code (online change) *)
		bInCopyCode : BOOL;
	END_VAR
END_METHOD


	(* Internal method *)
	{attribute 'hide'}
	METHOD FB_exit : BOOL
	VAR_INPUT
		(*  if TRUE, the exit method is called for exiting an instance that is copied afterwards (online change). *)
		bInCopyCode : BOOL;
	END_VAR
END_METHOD


	(* Set the normal vector of the disc. *)
	METHOD SetNormal
	VAR_IN_OUT
		(* The normal to set. *)
 {attribute 'GUID' := '8E451EF0-1EF7-2C22-40FE-C3C408FD9C3F'}
				normal : Tangent3D;
	END_VAR
END_METHOD


	(* Get the normal vector of the disc. *)
	METHOD GetNormal
	VAR
		(* The current normal vector of the disc. *)
 {attribute 'GUID' := '8E451EF0-1EF7-2C22-40FE-C3C408FD9C3F'}
				normal : Tangent3D;
	END_VAR
END_METHOD


	(* Get the area of the disc. *)
	METHOD GetArea : LREAL
END_METHOD


	PROPERTY radius : LREAL
GET
END_GET
SET
END_SET
END_PROPERTY

END_FUNCTION_BLOCK

// POUs/Shapes/Geometry3D/2D/Rectangle3D

	{attribute 'c++_compatible'}
	{attribute 'external_name' := 'Rectangle3D_GUID_6B770AE5_6A30_2E72_5ABD_A2AC23742091'}
	{attribute 'TcIecLibraryType'}
	{attribute 'no_explicit_call' :='do not call this POU directly'}
	{attribute 'no_assign'}
	FUNCTION_BLOCK Rectangle3D EXTENDS Geometry3D


	(* Internal method *)
	METHOD FB_init : BOOL
	VAR_INPUT
		(*  if TRUE, the retain variables are initialized (warm start / cold start) *)
		bInitRetains : BOOL;
		(*  if TRUE, the instance afterwards gets moved into the copy code (online change) *)
		bInCopyCode : BOOL;
	END_VAR
END_METHOD


	(* Internal method *)
	{attribute 'hide'}
	METHOD FB_exit : BOOL
	VAR_INPUT
		(*  if TRUE, the exit method is called for exiting an instance that is copied afterwards (online change). *)
		bInCopyCode : BOOL;
	END_VAR
END_METHOD


	(* Set the dimensions of the rectangle. *)
	METHOD SetDimensions
	VAR_INPUT
		(* The width of the rectangle to set. *)
		width : LREAL;
		(* The height of the rectangle to set. *)
		height : LREAL;
	END_VAR
END_METHOD


	(* Get the area of the rectangle. *)
	METHOD GetArea : LREAL
END_METHOD


	PROPERTY width : LREAL
GET
END_GET
SET
END_SET
END_PROPERTY


	PROPERTY height : LREAL
GET
END_GET
SET
END_SET
END_PROPERTY

END_FUNCTION_BLOCK

// POUs/Shapes/Geometry3D/3D/Sphere3D

	{attribute 'c++_compatible'}
	{attribute 'external_name' := 'Sphere3D_GUID_919F07C8_34AA_2B63_49DB_DC25375C40F3'}
	{attribute 'TcIecLibraryType'}
	{attribute 'no_explicit_call' :='do not call this POU directly'}
	{attribute 'no_assign'}
	FUNCTION_BLOCK Sphere3D EXTENDS Geometry3D


	(* Internal method *)
	METHOD FB_init : BOOL
	VAR_INPUT
		(*  if TRUE, the retain variables are initialized (warm start / cold start) *)
		bInitRetains : BOOL;
		(*  if TRUE, the instance afterwards gets moved into the copy code (online change) *)
		bInCopyCode : BOOL;
	END_VAR
END_METHOD


	(* Internal method *)
	{attribute 'hide'}
	METHOD FB_exit : BOOL
	VAR_INPUT
		(*  if TRUE, the exit method is called for exiting an instance that is copied afterwards (online change). *)
		bInCopyCode : BOOL;
	END_VAR
END_METHOD


	(* Get the volume of the sphere. *)
	METHOD GetVolume : LREAL
END_METHOD


	PROPERTY radius : LREAL
GET
END_GET
SET
END_SET
END_PROPERTY

END_FUNCTION_BLOCK

// POUs/Shapes/Geometry3D/3D/Cuboid3D

	{attribute 'c++_compatible'}
	{attribute 'external_name' := 'Cuboid3D_GUID_6385934B_4145_2D54_73FC_02FE0680C45B'}
	{attribute 'TcIecLibraryType'}
	{attribute 'no_explicit_call' :='do not call this POU directly'}
	{attribute 'no_assign'}
	FUNCTION_BLOCK Cuboid3D EXTENDS Geometry3D


	(* Internal method *)
	METHOD FB_init : BOOL
	VAR_INPUT
		(* if TRUE, the retain variables are initialized (warm start / cold start) *)
		bInitRetains : BOOL;
		(* if TRUE, the instance afterwards gets moved into the copy code (online change) *)
		bInCopyCode : BOOL;
	END_VAR
END_METHOD


	(* Internal method *)
	{attribute 'hide'}
	METHOD FB_exit : BOOL
	VAR_INPUT
		(* if TRUE, the exit method is called for exiting an instance that is copied afterwards (online change). *)
		bInCopyCode : BOOL;
	END_VAR
END_METHOD


	(* Set the dimensions of the cuboid. *)
	METHOD SetDimensions
	VAR_INPUT
		(* local x-component *)
		length : LREAL;
		(* local y-component *)
		width : LREAL;
		(* local z-component *)
		height : LREAL;
	END_VAR
END_METHOD


	(* Get the volume of the cuboid. *)
	METHOD GetVolume : LREAL
END_METHOD


	PROPERTY length : LREAL
GET
END_GET
SET
END_SET
END_PROPERTY


	PROPERTY width : LREAL
GET
END_GET
SET
END_SET
END_PROPERTY


	PROPERTY height : LREAL
GET
END_GET
SET
END_SET
END_PROPERTY

END_FUNCTION_BLOCK

// POUs/Shapes/Geometry3D/3D/Cylinder3D

	{attribute 'c++_compatible'}
	{attribute 'external_name' := 'Cylinder3D_GUID_071BC971_666D_25B6_6DAF_BC35272894FC'}
	{attribute 'TcIecLibraryType'}
	{attribute 'no_explicit_call' :='do not call this POU directly'}
	{attribute 'no_assign'}
	FUNCTION_BLOCK Cylinder3D EXTENDS Geometry3D


	(* Internal method *)
	METHOD FB_init : BOOL
	VAR_INPUT
		(* if TRUE, the retain variables are initialized (warm start / cold start) *)
		bInitRetains : BOOL;
		(* if TRUE, the instance afterwards gets moved into the copy code (online change) *)
		bInCopyCode : BOOL;
	END_VAR
END_METHOD


	(* Internal method *)
	{attribute 'hide'}
	METHOD FB_exit : BOOL
	VAR_INPUT
		(* if TRUE, the exit method is called for exiting an instance that is copied afterwards (online change). *)
		bInCopyCode : BOOL;
	END_VAR
END_METHOD


	(* Set the dimensions of the cylinder. *)
	METHOD SetDimensions
	VAR_INPUT
		(* The radius to set. *)
		radius : LREAL;
		(* The height to set. *)
		height : LREAL;
	END_VAR
END_METHOD


	(* Get the volume of the cylinder. *)
	METHOD GetVolume : LREAL
END_METHOD


	PROPERTY radius : LREAL
GET
END_GET
SET
END_SET
END_PROPERTY


	PROPERTY height : LREAL
GET
END_GET
SET
END_SET
END_PROPERTY

END_FUNCTION_BLOCK

// POUs/Shapes/Geometry3D/Functions/CheckCollision3D

	{attribute 'TcIecLibraryType'}
	{attribute 'external_name' := 'CheckCollision3D_GUID_64FBCBDA_0A11_2489_5600_BC7FA753EE69'}
	(* Check if two geometries are currently colliding. *)
	FUNCTION CheckCollision3D : BOOL
	VAR_IN_OUT
		geometry0	:	IPlcGeometry3D;	(* 1st input geometry to check for collision. *)
		geometry1	:	IPlcGeometry3D;	(* 2nd input geometry to check of collision. *)
	END_VAR

END_FUNCTION

// POUs/Shapes/Geometry3D/Functions/GetDistance3D

	{attribute 'TcIecLibraryType'}
	{attribute 'external_name' := 'GetDistance3D_GUID_9742F5CF_9DCB_238D_7937_6C271BFFBBD1'}
	(* Get the distance between two geometries. *)
	FUNCTION GetDistance3D : LREAL
	VAR_IN_OUT
		geometry0	:	IPlcGeometry3D;	(* 1st input geometry to calculate the distance of. *)
		geometry1	:	IPlcGeometry3D;	(* 2nd input geometry to calculate the distance of. *)
	END_VAR

END_FUNCTION

// POUs/Shapes/Geometry3D/Functions/GetLinkingLine3D

	{attribute 'TcIecLibraryType'}
	{attribute 'external_name' := 'GetLinkingLine3D_GUID_F47FFEC4_1D04_2C59_4AFA_05B1FB639013'}
	(* Get the shortest path between two geometries. *)
	FUNCTION GetLinkingLine3D : BOOL
	VAR_IN_OUT
		geometry0	:	IPlcGeometry3D;	(* 1st input geometry to calculate the linking line for. *)
		geometry1	:	IPlcGeometry3D;	(* 2nd input geometry to calculate the linking line for. *)
		linkingLine	:	Segment3D;	(* Return the resulting linking line. *)
	END_VAR

END_FUNCTION

// POUs/Shapes/Geometry3D/Functions/CreateIntersection2D

	{attribute 'TcIecLibraryType'}
	{attribute 'external_name' := 'CreateIntersection2D_GUID_C8A26629_EA38_2721_55D4_E819E42AF797'}
	(* Create a collection of intersections along a plane definition. *)
	FUNCTION CreateIntersection2D : BOOL
	VAR_IN_OUT
		container3D	:	Container3D;	(* Input container to create the intersections of. *)
		planeFrame	:	PositionSE3;	(* The coordinate frame to indicate the origin of the plane. *)
		container2D	:	Container2D;	(* Return the resulting collection of intersection. *)
	END_VAR

END_FUNCTION
